FUNCTION_BLOCK EL1808
VAR
	_io : EL1xx8_Data;
	{attribute addProperty Name "WcState"}
	_wcState : WcStateInputToggle;
	{attribute addProperty Name "Info data"}
	_infoData : InfoDataBase;
END_VAR

PROPERTY IO : REFERENCE TO EL1xx8_Data
GET
IO REF= _io;
END_GET
END_PROPERTY

PROPERTY WcState : REFERENCE TO WcStateInputToggle
GET
WcState REF= _wcState;
END_GET
END_PROPERTY

END_FUNCTION_BLOCK

(* stored: Version 1.1.0.1, ProductVersion 3.1.4024.9
   POU EL1808: Id {6b4f7620-935f-0051-0611-6de329f434af}, SpecialFunc None
   Property IO: Id {7a7296ca-2938-044d-335b-de86b53e978a}
   Get Get: Id {1e1ecf8c-811c-004e-0092-8681ced56b5e}
   Property WcState: Id {71aa7a32-85df-0034-0e88-42da49b30250}
   Get Get: Id {34b6d9f6-836e-0305-0cc9-4405539df2c4} *)
